FUNCTION_BLOCK IO_READER
  (* Version 1.0, 2005-06-27, Goran Cengic, Chalmers *)
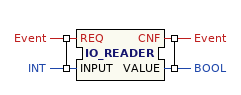
  EVENT_INPUT
    REQ WITH INPUT;
  END_EVENT
  EVENT_OUTPUT
    CNF WITH VALUE;
  END_EVENT
  VAR_INPUT
    INPUT : INT; (* The number of the input pin to read from the digital I/O card. *)
  END_VAR
  VAR_OUTPUT
    VALUE : BOOL; (* The value read from the digital I/O card. *)
  END_VAR
END_FUNCTION_BLOCK
